PROGRAM HMI
VAR
	displayvalues		: ARRAY[1..25] OF ST_DisplayPositions;
	displaycounter		: INT:=1;
	insidelimits		: BOOL:= FALSE;
	bLoadOK				: BOOL:= FALSE;
	bLoaded				: BOOL:= FALSE;
	bUnload				: BOOL:= FALSE;
	bTgtLoaded			: BOOL:= FALSE;
	bEditEnable			: BOOL:= FALSE;
	DisplayTgtPos	:	STRING:= '';	
	
//Indicator Flags	
	bSoftUpLimFlag		: BOOL;
	bSoftDownLimFlag	: BOOL;
	bSoftLimFlag		: BOOL;
	bLimitHeaderFlag	: BOOL;
	bSystemFlag			: BOOL:= FALSE;
		
//Color Fields
	dwUpArrow			: DWORD;
	dwDownArrow			: DWORD;
	dwDoorFlag			: DWORD;
	dwDoor1				: DWORD;
	dwDoor2				: DWORD;
	dwDoor3				: DWORD;
	dwDoor4				: DWORD;
	dwCrushFlag			: DWORD;
	dwSysFaultFlag		: DWORD;

END_VAR

//Displayed Values Logic
	CASE displaycounter OF
	1..25: (* Creates a state machine that will write XML values to displayed values *)
		IF 	XML.savedvalues.SavedPos[displaycounter].targetclear = FALSE THEN 
			displayvalues[displaycounter].target := '';
			//displayvalues[displaycounter].description := '';
		ELSE	
			displayvalues[displaycounter].target := CONCAT((REAL_TO_STRING(XML.savedvalues.SavedPos[displaycounter].target)),'"');
		END_IF
		displaycounter := displaycounter +1;
	26: (*Resets State Machine *)
			displaycounter := 1;
	END_CASE
	
	displayvalues[displaycounter].description := (XML.savedvalues.SavedPos[displaycounter].description);	
	
//Determines if Target is inside Soft Limits
	IF XML.savedvalues.savedpos[GV_HMI.RowSelect].target <= (XML.savedvalues.UpSoftLim) AND XML.savedvalues.savedpos[GV_HMI.RowSelect].target >= (XML.savedvalues.DownSoftLim) THEN
		insidelimits := TRUE;
	ELSE
		insidelimits := FALSE;
	END_IF
	
//Load Button Logic
	IF XML.savedvalues.savedpos[GV_HMI.RowSelect].targetclear AND insidelimits AND GV_LIFT.RUN_BUTTON_OUT THEN
		bLoadOK	:= TRUE;
	ELSE
		bLoadOK	:= FALSE;	
	END_IF

//Removing Target if highlighted target changes
	IF xml.savedvalues.SavedPos[GV_HMI.RowSelected].target <> xml.savedvalues.SavedPos[GV_HMI.RowSelect].target THEN
		bTgtLoaded := FALSE;
	END_IF
	
// Displaying Loaded Target
	IF 	bTgtLoaded = FALSE OR bLoadOK = FALSE OR GV_LIFT.MTS_ALLOWED = FALSE THEN
		DisplayTgtPos:= '';
	ELSE
		DisplayTgtPos:= CONCAT(REAL_TO_STRING((GV_LIFT.TARGET_POSITION)),'"');
	END_IF

// Hiding load Button to Display Unload Button
	IF bLoadOK = TRUE AND bTgtLoaded = TRUE AND GV_LIFT.MTS_ALLOWED THEN
		bUnload := TRUE;
	ELSE bUnload := FALSE;	
	END_IF

//System Indicator

//Soft Up Limit Indicator
	IF (GV_LIFT.CURRENT_POSITION > XML.savedvalues.UpSoftLim) AND NOT GV_LIFT.LIMIT_OVERRIDE_BUTTON_IN THEN
		bSoftUpLimFlag := FALSE;
	ELSE bSoftUpLimFlag := TRUE;
	END_IF
	
//Soft Down Limit Indicator
	IF (GV_LIFT.CURRENT_POSITION < XML.savedvalues.DownSoftLim) AND NOT GV_LIFT.LIMIT_OVERRIDE_BUTTON_IN THEN
		bSoftDownLimFlag := FALSE;
	ELSE bSoftDownLimFlag := TRUE;
	END_IF
		
//Soft Limit System Indicator
	IF (GV_LIFT.CURRENT_POSITION < XML.savedvalues.DownSoftLim) OR (GV_LIFT.CURRENT_POSITION < XML.savedvalues.UpSoftLim) OR GV_LIFT.LIMIT_OVERRIDE_BUTTON_IN THEN
		bSoftLimFlag := TRUE;
		bSystemFlag:= TRUE;
	ELSE bSoftLimFlag := FALSE;
	END_IF
	
//Limit Safety Page Header
	IF NOT bSoftLimFlag OR NOT GV_LIFT.UP_LIMIT_INDICATOR_IN OR NOT GV_LIFT.DOWN_LIMIT_INDICATOR_IN OR NOT GV_LIFT.ULTIMATE_LIMIT_INDICATOR_IN THEN
		bLimitHeaderFlag := FALSE;
	ELSE bLimitHeaderFlag := TRUE;
	END_IF
 	

//Button and Inidcator Calls
	HMI_Up_Arrow_Indicator();
	HMI_Down_Arrow_Indicator();
	HMI_Door_Toggle();
	HMI_Crush_Indicator();
	HMI_System_Indicator();
	HMI_Hard_Limits();
	HMI_Ultimate_Limit();

END_PROGRAM

(* stored: Version 1.1.0.1, ProductVersion 3.1.4022.12
   POU HMI: Id {64e13a00-698b-4f83-9fef-3d94ef99aec6}, SpecialFunc None *)
